// Mitsubishi GX Works2 project: XOR   PLC: Q03UDV

PROGRAM MAIN
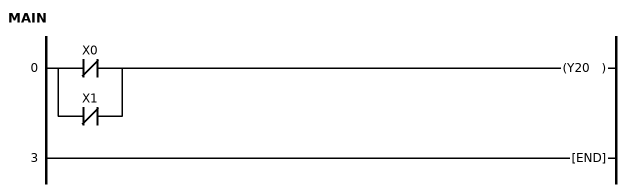
0     LDI     X0
      ORI     X1
      OUT     Y20
3     END
END_PROGRAM
